Staubli VAL3: setLanguage.pgx

public program setLanguage(string x_sPath)
  local num l_nResult
  local string l_sMessage
begin
  //
  call language:message(l_sMessage,-7)
  l_nResult=language:libLoad(x_sPath)
  delay(0)
  if l_nResult!=0
    popUpMsg(l_sMessage+x_sPath+" ; "+toString("",l_nResult))
  endIf
end
